TYPE AxesAlphaUnits :
(
	HOURS := 0,
	DEGREES := 1,
	RADIANS := 2
);
END_TYPE

(* stored: Version 1.1.0.1, ProductVersion 3.1.4019.2
   DUT AxesAlphaUnits: Id {f62da930-4441-4829-a00a-027e64bec041} *)
